FUNCTION_BLOCK FB_StringBuilder
VAR
	sContent : STRING; // Store temporary strings;
END_VAR

METHOD Append : POINTER TO FB_StringBuilder
VAR_INPUT
	sText : STRING;
END_VAR
sContent := CONCAT(STR1 := sContent, STR2 := sText);
Append := THIS;
END_METHOD

METHOD Clear : POINTER TO FB_StringBuilder
VAR_INPUT
END_VAR
sContent := '';
Clear := THIS;
END_METHOD

METHOD ToString : STRING
VAR_INPUT
END_VAR
ToString := sContent; // return internal content
END_METHOD

END_FUNCTION_BLOCK

(* stored: Version 1.1.0.1, ProductVersion 3.1.4024.12
   POU FB_StringBuilder: Id {9b7d1f4b-176f-41d4-8627-3b0bc05f09de}, SpecialFunc None
   Method Append: Id {bbe18d8f-884b-4ab2-a1d1-84173cab1b17}
   Method Clear: Id {a2db7a52-3431-4f44-a4f6-d74064bb23ba}
   Method ToString: Id {6bddf2a5-309c-4a77-8635-15b0db2737b5} *)
